FUNCTION_BLOCK F_TAN (* tangent in radians *)
  PACKAGE iec61131::numerical;
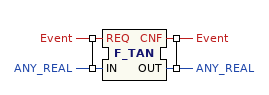
  EVENT_INPUT
    REQ WITH IN; (* Service Request *)
  END_EVENT
  EVENT_OUTPUT
    CNF WITH OUT; (* Confirmation of Requested Service *)
  END_EVENT
  VAR_INPUT
    IN : ANY_REAL; (* Event Input Qualifier *)
  END_VAR
  VAR_OUTPUT
    OUT : ANY_REAL; (* Event Output Qualifier *)
  END_VAR
END_FUNCTION_BLOCK
